(* PLC project SafeLOGIC-1, BrAutomation SafeDESIGNER  5.15.0.0 *)
(* stored: companyURL http://www.br-automation.com, creationDateTime Thu Jan 06 17:36:35 2022 *)

PROGRAM Decode

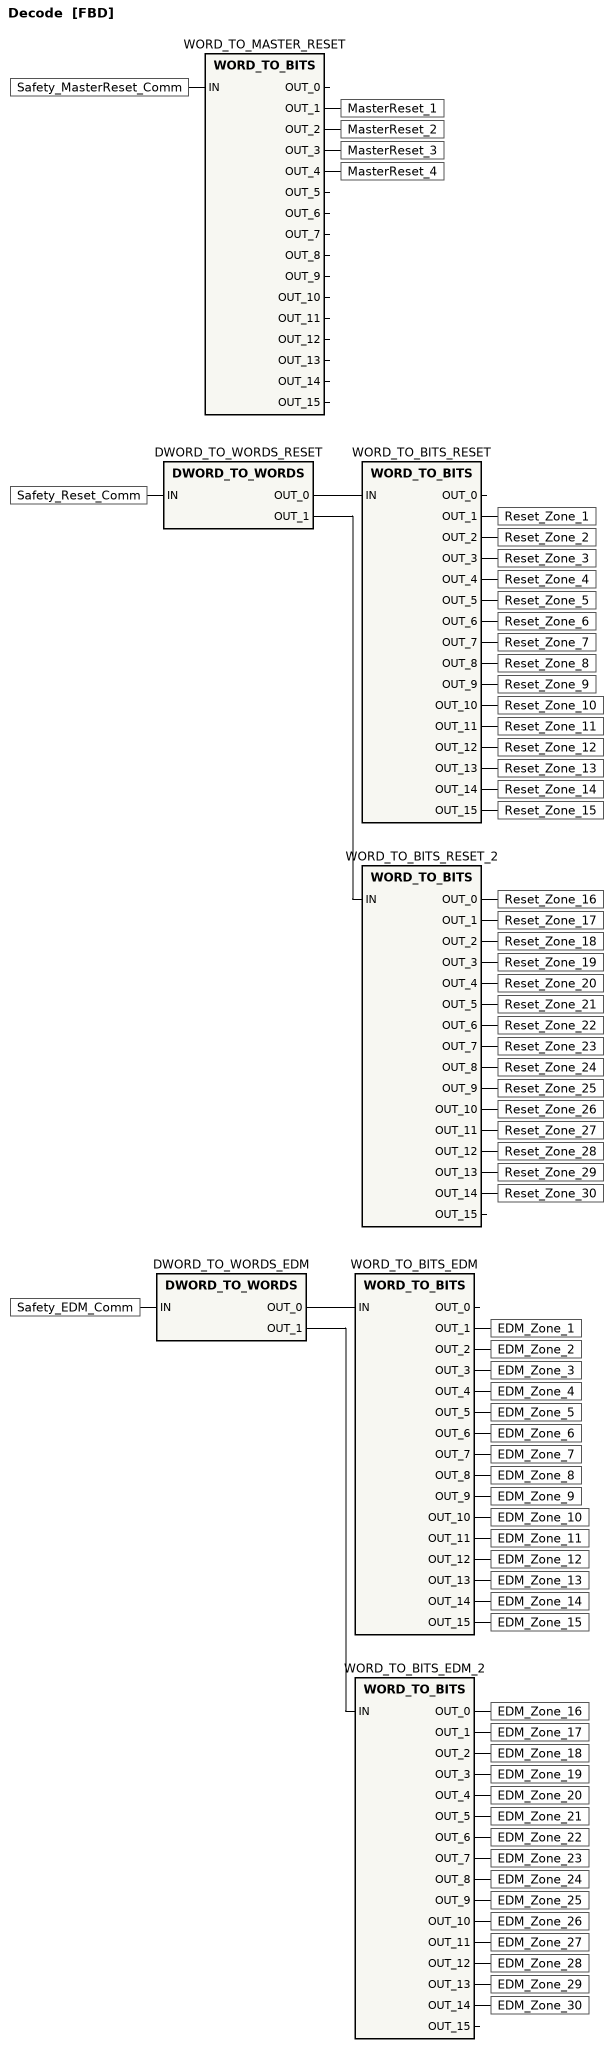
(* FBD diagram, written out as Structured Text *)
WORD_TO_MASTER_RESET(IN := Safety_MasterReset_Comm);
MasterReset_1 := WORD_TO_MASTER_RESET.OUT_1;
MasterReset_2 := WORD_TO_MASTER_RESET.OUT_2;
MasterReset_3 := WORD_TO_MASTER_RESET.OUT_3;
MasterReset_4 := WORD_TO_MASTER_RESET.OUT_4;
DWORD_TO_WORDS_RESET(IN := Safety_Reset_Comm);
WORD_TO_BITS_RESET(IN := DWORD_TO_WORDS_RESET.OUT_0);
Reset_Zone_1 := WORD_TO_BITS_RESET.OUT_1;
Reset_Zone_4 := WORD_TO_BITS_RESET.OUT_4;
Reset_Zone_2 := WORD_TO_BITS_RESET.OUT_2;
Reset_Zone_5 := WORD_TO_BITS_RESET.OUT_5;
Reset_Zone_3 := WORD_TO_BITS_RESET.OUT_3;
Reset_Zone_6 := WORD_TO_BITS_RESET.OUT_6;
Reset_Zone_7 := WORD_TO_BITS_RESET.OUT_7;
Reset_Zone_10 := WORD_TO_BITS_RESET.OUT_10;
Reset_Zone_11 := WORD_TO_BITS_RESET.OUT_11;
Reset_Zone_9 := WORD_TO_BITS_RESET.OUT_9;
Reset_Zone_8 := WORD_TO_BITS_RESET.OUT_8;
Reset_Zone_12 := WORD_TO_BITS_RESET.OUT_12;
Reset_Zone_15 := WORD_TO_BITS_RESET.OUT_15;
Reset_Zone_13 := WORD_TO_BITS_RESET.OUT_13;
Reset_Zone_14 := WORD_TO_BITS_RESET.OUT_14;
WORD_TO_BITS_RESET_2(IN := DWORD_TO_WORDS_RESET.OUT_1);
Reset_Zone_16 := WORD_TO_BITS_RESET_2.OUT_0;
Reset_Zone_17 := WORD_TO_BITS_RESET_2.OUT_1;
Reset_Zone_18 := WORD_TO_BITS_RESET_2.OUT_2;
Reset_Zone_19 := WORD_TO_BITS_RESET_2.OUT_3;
Reset_Zone_20 := WORD_TO_BITS_RESET_2.OUT_4;
Reset_Zone_21 := WORD_TO_BITS_RESET_2.OUT_5;
Reset_Zone_22 := WORD_TO_BITS_RESET_2.OUT_6;
Reset_Zone_23 := WORD_TO_BITS_RESET_2.OUT_7;
Reset_Zone_24 := WORD_TO_BITS_RESET_2.OUT_8;
Reset_Zone_25 := WORD_TO_BITS_RESET_2.OUT_9;
Reset_Zone_26 := WORD_TO_BITS_RESET_2.OUT_10;
Reset_Zone_27 := WORD_TO_BITS_RESET_2.OUT_11;
Reset_Zone_28 := WORD_TO_BITS_RESET_2.OUT_12;
Reset_Zone_29 := WORD_TO_BITS_RESET_2.OUT_13;
Reset_Zone_30 := WORD_TO_BITS_RESET_2.OUT_14;
DWORD_TO_WORDS_EDM(IN := Safety_EDM_Comm);
WORD_TO_BITS_EDM(IN := DWORD_TO_WORDS_EDM.OUT_0);
EDM_Zone_1 := WORD_TO_BITS_EDM.OUT_1;
EDM_Zone_2 := WORD_TO_BITS_EDM.OUT_2;
EDM_Zone_3 := WORD_TO_BITS_EDM.OUT_3;
EDM_Zone_4 := WORD_TO_BITS_EDM.OUT_4;
EDM_Zone_5 := WORD_TO_BITS_EDM.OUT_5;
EDM_Zone_6 := WORD_TO_BITS_EDM.OUT_6;
EDM_Zone_7 := WORD_TO_BITS_EDM.OUT_7;
EDM_Zone_8 := WORD_TO_BITS_EDM.OUT_8;
EDM_Zone_9 := WORD_TO_BITS_EDM.OUT_9;
EDM_Zone_10 := WORD_TO_BITS_EDM.OUT_10;
EDM_Zone_11 := WORD_TO_BITS_EDM.OUT_11;
EDM_Zone_12 := WORD_TO_BITS_EDM.OUT_12;
EDM_Zone_13 := WORD_TO_BITS_EDM.OUT_13;
EDM_Zone_14 := WORD_TO_BITS_EDM.OUT_14;
EDM_Zone_15 := WORD_TO_BITS_EDM.OUT_15;
WORD_TO_BITS_EDM_2(IN := DWORD_TO_WORDS_EDM.OUT_1);
EDM_Zone_16 := WORD_TO_BITS_EDM_2.OUT_0;
EDM_Zone_17 := WORD_TO_BITS_EDM_2.OUT_1;
EDM_Zone_18 := WORD_TO_BITS_EDM_2.OUT_2;
EDM_Zone_19 := WORD_TO_BITS_EDM_2.OUT_3;
EDM_Zone_20 := WORD_TO_BITS_EDM_2.OUT_4;
EDM_Zone_21 := WORD_TO_BITS_EDM_2.OUT_5;
EDM_Zone_22 := WORD_TO_BITS_EDM_2.OUT_6;
EDM_Zone_23 := WORD_TO_BITS_EDM_2.OUT_7;
EDM_Zone_24 := WORD_TO_BITS_EDM_2.OUT_8;
EDM_Zone_25 := WORD_TO_BITS_EDM_2.OUT_9;
EDM_Zone_26 := WORD_TO_BITS_EDM_2.OUT_10;
EDM_Zone_27 := WORD_TO_BITS_EDM_2.OUT_11;
EDM_Zone_28 := WORD_TO_BITS_EDM_2.OUT_12;
EDM_Zone_29 := WORD_TO_BITS_EDM_2.OUT_13;
EDM_Zone_30 := WORD_TO_BITS_EDM_2.OUT_14;
END_PROGRAM
